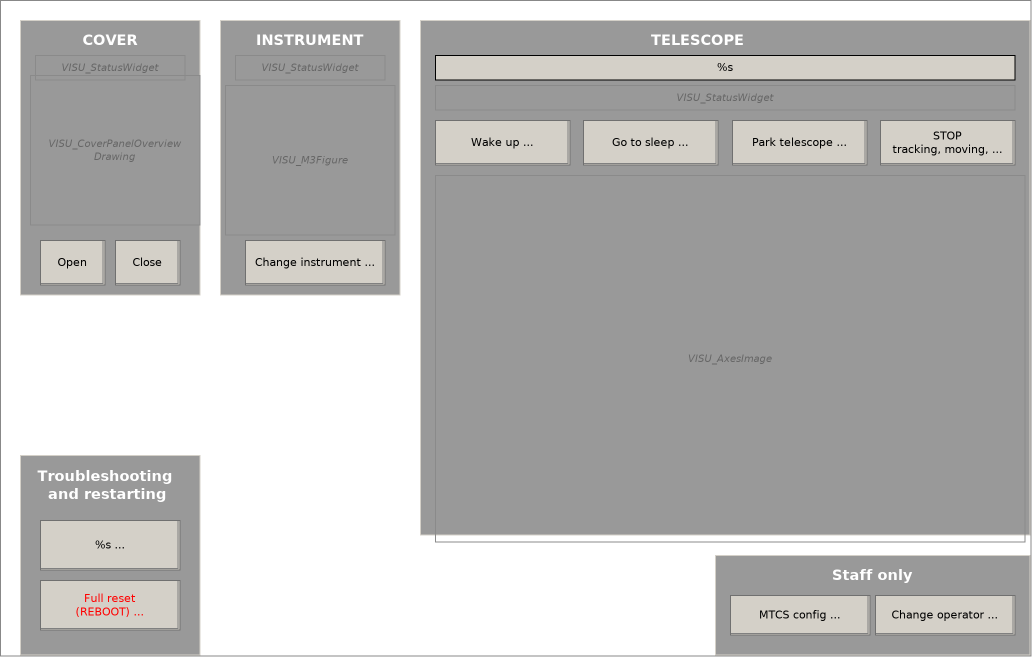
VISUALIZATION VISU_MTCSHome  // 1032x657
VAR_IN_OUT
	mtcs : MTCS;
	mtcsWidget : MTCSWidget;	
END_VAR
    Rectangle (220,20 180x275)
    Rectangle (20,20 180x275)
    Frame (30,75 170x150)
        shows VISU_CoverPanelOverviewDrawing(cover := mtcs.parts.cover, coverWidget := mtcsWidget.cover)
    Label (35,25 150x30), "COVER"
    Button (40,240 65x45), "Open", input disabled if: mtcs.parts.cover.processes.open.statuses.enabledStatus.disabled
        OnMouseClick: execute { mtcs.parts.cover.processes.open.do_request := TRUE; }
    Button (115,240 65x45), "Close", input disabled if: mtcs.parts.cover.processes.close.statuses.enabledStatus.disabled
        OnMouseClick: execute { mtcs.parts.cover.processes.close.do_request := TRUE; }
    Label (235,25 150x30), "INSTRUMENT"
    Frame (225,85 170x150)
        shows VISU_M3Figure(m3 := mtcs.parts.m3, widget := mtcsWidget.m3, hideDetails := mtcsWidget.hideDetails)
    Frame (35,55 150x25)
        shows VISU_StatusWidget(widget := mtcsWidget.cover.actualStatus)
    Frame (235,55 150x25)
        shows VISU_StatusWidget(widget := mtcsWidget.changeInstrumentStatus)
    Rectangle (715,555 315x100)
    Label (715,560 315x30), "Staff only"
    Button (730,595 140x40), "MTCS config ...", input disabled if: NOT mtcs.statuses.operatorStatus.tech
        OnMouseClick: OpenDialog Dialog=VISU_MTCSConfigDialog, OpenModal=True, OpenCentered=True
    Rectangle (420,20 610x515)
    Label (435,25 525x30), "TELESCOPE"
    Button (583,120 135x45), "Go to sleep ...", input disabled if: mtcs.processes.goToSleep.statuses.enabledStatus.disabled
        OnMouseClick: OpenDialog Dialog=VISU_MTCSGoToSleepDialog, OpenModal=True, OpenCentered=True
    Button (435,120 135x45), "Wake up ...", input disabled if: mtcs.processes.wakeUp.statuses.enabledStatus.disabled
        OnMouseClick: OpenDialog Dialog=VISU_MTCSWakeUpTelescopeDialog, OpenModal=True, OpenCentered=True
    Rectangle (20,455 180x200)
    Label (35,460 145x50), "Troubleshooting and restarting"
    Button (40,580 140x50), "Full reset (REBOOT) ..."
        OnMouseClick: OpenDialog Dialog=VISU_MTCSRebootDialog, OpenModal=True, OpenCentered=True
    Button (40,520 140x50), "%s ...", text variable: mtcsWidget.button_initialize.textOneLine, input disabled if: mtcsWidget.button_initialize.deactivate
        OnMouseClick: OpenDialog Dialog=VISU_MTCSInitializeDialog, OpenModal=True, OpenCentered=True
    Button (875,595 140x40), "Change operator ..."
        OnMouseClick: OpenDialog Dialog=VISU_MTCSChangeOperatorDialog, OpenModal=True, OpenCentered=True
    Button (245,240 140x45), "Change instrument ..."
        OnMouseClick: OpenDialog Dialog=VISU_MTCSChangeInstrumentDialog, OpenModal=True, OpenCentered=True
    Button (732,120 135x45), "Park telescope ..."
        OnMouseClick: OpenDialog Dialog=VISU_MTCSParkTelescopeDialog, OpenModal=True, OpenCentered=True
    Frame (435,175 590x367)
        shows VISU_AxesImage(ref := mtcs.parts.axes, widget := mtcsWidget.axes)
    Button (880,120 135x45), "STOP tracking, moving, ...", input disabled if: mtcs.parts.axes.processes.stop.statuses.enabledStatus.disabled
        OnMouseClick: execute { mtcs.parts.axes.processes.stop.request(); }
    Frame (435,85 580x25)
        shows VISU_StatusWidget(widget := mtcsWidget.axes.actualStatus)
    Rectangle (435,55 580x25), "%s", text variable: mtcsWidget.activityStatus.description, colour variable: mtcsWidget.activityStatus.bgColor
        p55702900: mtcsWidget.activityStatus.fgColor
        p3450524324: mtcsWidget.activityStatus.fgColor
END_VISUALIZATION

(* stored: Version 1.1.0.1, ProductVersion 3.1.4019.2
   Visu VISU_MTCSHome: Id {493d4f04-6425-4c51-8a28-dbdb37752d5c} *)
